(* IEC 61131-3 sources: POMIRTS_lab3/AS/Library/MTSystem/V1.00.1, 3 files *)

(* ---- MTSystem.typ ---- *)
(********************************************************************
 * COPYRIGHT -- Bernecker + Rainer
 ********************************************************************
 * Library: MTSystem
 * File: MTSystem.typ
 * Author: B&R
 * Created: July 2013
 ********************************************************************
 * Data types of library XXTemplate
 ********************************************************************)

TYPE
	MTSystemBodeInternalType : 	STRUCT
		NbValidExtSystemReferences : USINT; (*Data for internal use.*)
		UpdateOld : BOOL; (*Data for internal use.*)
		EnableOld : BOOL; (*Data for internal use.*)
		ParametersValid : BOOL; (*Data for internal use.*)
		CalcPlotData : BOOL; (*Data for internal use.*)
		CalcPlotDataOld : BOOL; (*Data for internal use.*)
		CalcFrequencyData : BOOL; (*Data for internal use.*)
		CalcFrequencyDataOld : BOOL; (*Data for internal use.*)
		RunCalculation : BOOL; (*Data for internal use.*)
		MinFrequency : REAL; (*Data for internal use.*)
		MaxFrequency : REAL; (*Data for internal use.*)
		Frequency : REAL; (*Data for internal use.*)
	END_STRUCT;
	MTSystemBode2InternalType : 	STRUCT
		NbValidExtSystemReferences : USINT; (*Data for internal use.*)
		CalcPlotData : BOOL; (*Data for internal use.*)
		CalcPlotDataOld : BOOL; (*Data for internal use.*)
		EnableOld : BOOL; (*Data for internal use.*)
	END_STRUCT;
	MTSystemTransferFcnInternalType : 	STRUCT
		CycleTime : REAL; (*Task cycle time. Unit: [s].*)
		UpdateOld : BOOL; (*Data for internal use.*)
		EnableOld : BOOL; (*Data for internal use.*)
		EnableDone : BOOL; (*Data for internal use.*)
		DisabledBusy : USINT; (*Data for internal use.*)
		ParametersValid : BOOL; (*Data for internal use.*)
		SampleTime : REAL; (*Data for internal use.*)
		SysRefParaNew : BOOL; (*Data for internal use.*)
		CounterOld : UDINT; (*Data for internal use.*)
		Order : USINT; (*Data for internal use.*)
		PresetOK : BOOL; (*Data for internal use.*)
		PresetCoefficients : LREAL; (*Data for internal use.*)
		BVector : ARRAY[0..5]OF LREAL; (*Data for internal use.*)
		AVector : ARRAY[0..5]OF LREAL; (*Data for internal use.*)
		XVector : ARRAY[0..4]OF LREAL; (*Data for internal use.*)
		OutPresetValue : REAL; (*Data for internal use.*)
		SetOut : BOOL; (*Data for internal use.*)
		SetOutOld : BOOL; (*Data for internal use.*)
		SystemReference : MTTransferFcnType; (*Data for internal use.*)
	END_STRUCT;
END_TYPE

(* ---- MTSystem.fun ---- *)
(********************************************************************
 * COPYRIGHT -- Bernecker + Rainer
 ********************************************************************
 * Library: MTSystem
 * File: MTSystem.fun
 * Author: B&R
 * Created: July 2013
 ********************************************************************
 * Functions and function blocks of library XXTemplate
 ********************************************************************)

FUNCTION_BLOCK MTSystemTransferFcn (*This function block implements a general continuous transfer function G(s). Optional it is possible to implement a discrete transfer function G(z) with DiscreteSampleTime > 0.*)
	VAR_INPUT
		Enable : BOOL; (*Enable function block.*) (* *) (*#PAR#*)
		Numerator : ARRAY[0..5] OF REAL; (*Coefficients of numerator [b0, b1, b2, ... bn].*) (* *) (*#PAR#*)
		Denominator : ARRAY[0..5] OF REAL; (*Coefficients of denominator [a0, a1, a2, ... an].*) (* *) (*#PAR#*)
		SampleTime : REAL; (*SampleTime = 0 (default) ... continuous transfer function. DiscreteSampleTime > 0 ... discrete transfer function.*) (* *) (*#PAR#*)
		Update : BOOL; (*Parameters update trigger.*) (* *) (*#PAR#*)
		In : REAL; (*Input variable.*) (* *) (*#CYC#*)
		OutPresetValue : REAL; (*Preset value for Out.*) (* *) (*#CMD#OPT#*)
		SetOut : BOOL; (*Sets Out to OutPresetValue on rising edge.*) (* *) (*#CMD#OPT#*)
	END_VAR
	VAR_OUTPUT
		Busy : BOOL; (*Function block is working.*) (* *) (*#PAR#*)
		Active : BOOL; (*Function block is active.*) (* *) (*#PAR#*)
		Error : BOOL; (*Indicates an error.*) (* *) (*#PAR#*)
		StatusID : DINT; (*Status information.*) (* *) (*#PAR#*)
		UpdateDone : BOOL; (*Update is sucessful.*) (* *) (*#PAR#*)
		Out : REAL; (*Output variable.*) (* *) (*#CYC#*)
		SystemReference : UDINT; (*System reference.*) (* *) (*#CMD#OPT#*)
	END_VAR
	VAR
		Internal : MTSystemTransferFcnInternalType; (*Data for internal use.*)
	END_VAR
END_FUNCTION_BLOCK

FUNCTION_BLOCK MTSystemBode (*This function block gives the amplitude and phase response of a specified system.*)
	VAR_INPUT
		Enable : BOOL; (*Enable/disable function block.*) (* *) (*#PAR#*)
		SystemReference : ARRAY[0..2] OF UDINT; (*System reference.*) (* *) (*#CMD#*)
		MinFrequency : REAL; (*Minimum frequency in Hz.*) (* *) (*#CMD#OPT#*)
		CalcPlotData : BOOL; (*Calculate bode plot data on rising edge.*) (* *) (*#CMD#*)
		Frequency : REAL; (*Frequency at which magnitude and phase response is required in Hz.*) (* *) (*#CMD#OPT#*)
		CalcFrequencyData : BOOL; (*Calculate magnitude and phase on rising edge at specified frequency.*) (* *) (*#CMD#OPT#*)
	END_VAR
	VAR_OUTPUT
		Active : BOOL; (*Function block is active.*) (* *) (*#PAR#*)
		Error : BOOL; (*Indicates an error.*) (* *) (*#PAR#*)
		StatusID : DINT; (*Status information.*) (* *) (*#PAR#*)
		CalcPlotDataDone : BOOL; (*Calculation of plot data done.*) (* *) (*#CMD#*)
		PlotData : MTBodeType; (*Bode plot data.*) (* *) (*#CMD#*)
		CalcFrequencyDataDone : BOOL; (*Calculation of frequency data done.*) (* *) (*#CMD#OPT#*)
		Magnitude : REAL; (*Magnitude at specified frequency.*) (* *) (*#CMD#OPT#*)
		Phase : REAL; (*Phase at specified frequency.*) (* *) (*#CMD#OPT#*)
	END_VAR
	VAR
		Internal : MTSystemBodeInternalType; (*Data for internal use.*)
	END_VAR
END_FUNCTION_BLOCK

(* ---- MTSystem.var ---- *)
(********************************************************************
 * COPYRIGHT -- Bernecker + Rainer
 ********************************************************************
 * Library: MTSystem
 * File: MTSystem.var
 * Author: B&R
 * Created: August, 2013
 ********************************************************************
 * Constants of library XXTemplate
 ********************************************************************)
VAR CONSTANT
	mtACD_ERR_DATA_NOT_AVAILABLE : DINT := -1058013183; (*Error: The data in the system reference is invalid.*)
	mtACD_ERR_SYSTEM_TYPE_INVALID : DINT := -1058013182; (*Error: The system type specified in the system reference is invalid.*)
	mtACD_ERR_DISCR_SAMPLE_TIME_NEG : DINT := -1058011184; (*Error: Sample time is negative.*)
	mtACD_ERR_TF_ORDER_NOT_MINIMAL : DINT := -1058011183; (*Error: Order of transfer function not minimal.*)
	mtACD_ERR_WRONG_TASK_CLASS : DINT := -1058011182; (*Error: Incorrect task class. Task cyclic time is not the same as sample time.*)
	mtACD_ERR_DENOM_COEFF_INVALID : DINT := -1058011181; (*Error: Denominator coefficient Denominator[Order] is 0.*)
	mtACD_ERR_FREQUENCY_INVALID : DINT := -1058011180; (*Error: Frequency is invalid.*)
	mtACD_ERR_INVALID_SYSREF : DINT := -1058011179; (*Error: System referemce is invalid.*)
	mtACD_ERR_NO_COMMON_FREQ_ZONE : DINT := -1058011178; (*Error: No common frequency zone is available.*)
	mtACD_WRN_OTHER_FB_USES_SYSREF : DINT := -2131755008; (*Warning: Another function block is using the data for this system reference.*)
	mtACD_WRN_DISCR_SAMPLE_TIME_NEG : DINT := -2131753008; (*Warning: SamplingTime is invalid. Retaining the last valid configuration.*)
	mtACD_WRN_TF_ORDER_NOT_MINIMAL : DINT := -2131753007; (*Warning: Order is not minimal. Retaining the last valid configuration.*)
	mtACD_WRN_TF_PRESET_INVALID : DINT := -2131753006; (*Warning: The preset output value is invalid.*)
	mtACD_WRN_DENOM_COEFF_INVALID : DINT := -2131753005; (*Warning: Denominator coefficients are zero. Retaining the last valid configuration.*)
	mtACD_WRN_FREQ_RANGE_INVALID : DINT := -2131753003; (*Warning: MaxFrequency is outside the permitted range (4 decades). The last value of the frequency domain will be used for MaxFrequency.*)
END_VAR
